{attribute 'linkalways'} 
{attribute 'no_explicit_call' := 'This FB is a CLASS and must be accessed using methods or properties'}
{attribute 'enable_dynamic_creation'}
FUNCTION_BLOCK DefaultHomingBuilder IMPLEMENTS I_HomingBuilder, I_PositioningHomingBuilder, I_DefaultHomingBuilder
VAR
	_axis : I_Axis;
	_position : LREAL;
	_options : ST_HomingOptions;
	_cam : REFERENCE TO BOOL;
END_VAR

METHOD BuildDefaultHomingCommand : I_HomingCommand
VAR
	pCmd : POINTER TO HomingCommand;
	cmd : I_HomingCommand;
END_VAR
pCmd := __NEW(HomingCommand(
	axis := _axis,
	position := _position,
	mode := HomingMode.Default,
	options := _options,
	cam := _cam
));
BuildDefaultHomingCommand := pCmd^;
END_METHOD

METHOD BuildDirectHomingCommand : I_HomingCommand
VAR
	pCmd : POINTER TO HomingCommand;
	cmd : I_HomingCommand;
	null : BOOL;
END_VAR
pCmd := __NEW(HomingCommand(
	axis := _axis,
	position := _position,
	mode := HomingMode.Direct,
	options := _options,
	cam := null
));
BuildDirectHomingCommand := pCmd^;
END_METHOD

METHOD BuildForceCalibrationCommand : I_HomingCommand
VAR
	pCmd : POINTER TO HomingCommand;
	cmd : I_HomingCommand;
	null : BOOL;
END_VAR
pCmd := __NEW(HomingCommand(
	axis := _axis,
	position := _position,
	mode := HomingMode.ForceCalibration,
	options := _options,
	cam := null
));
BuildForceCalibrationCommand := pCmd^;
END_METHOD

METHOD BuildResetCalibrationCommand : I_HomingCommand
VAR
	pCmd : POINTER TO HomingCommand;
	cmd : I_HomingCommand;
	null : BOOL;
END_VAR
pCmd := __NEW(HomingCommand(
	axis := _axis,
	position := _position,
	mode := HomingMode.ResetCalibration,
	options := _options,
	cam := null
));
BuildResetCalibrationCommand := pCmd^;
END_METHOD

METHOD Cam : I_DefaultHomingBuilder
VAR_INPUT
	value : REFERENCE TO BOOL;
END_VAR
_cam REF= value;
Cam := THIS^;
END_METHOD

METHOD ClearLag : I_PositioningHomingBuilder
_options.ClearPositionLag := TRUE;
ClearLag := THIS^;
END_METHOD

METHOD FB_init : BOOL
VAR_INPUT
	bInitRetains : BOOL; // if TRUE, the retain variables are initialized (warm start / cold start)
	bInCopyCode : BOOL;  // if TRUE, the instance afterwards gets moved into the copy code (online change)
	axis : I_Axis;
END_VAR
_axis := axis;
END_METHOD

METHOD KeepLag : I_PositioningHomingBuilder
_options.ClearPositionLag := FALSE;
KeepLag := THIS^;
END_METHOD

METHOD Position : I_PositioningHomingBuilder
VAR_INPUT
	value : LREAL;
END_VAR
_position := value;
Position := THIS^;
END_METHOD

METHOD ReferenceMode : I_DefaultHomingBuilder
VAR_INPUT
	value : EncoderReferenceMode;
END_VAR
_options.ReferenceMode := value;
ReferenceMode := THIS^;
END_METHOD

METHOD SearchDirection : I_DefaultHomingBuilder
VAR_INPUT
	value : Direction;
END_VAR
_options.SearchDirection := value;
SearchDirection := THIS^;
END_METHOD

METHOD SearchVelocity : I_DefaultHomingBuilder
VAR_INPUT
	value	: LREAL;
END_VAR
_options.SearchVelocity := value;
SearchVelocity := THIS^;
END_METHOD

METHOD SyncDirection : I_DefaultHomingBuilder
VAR_INPUT
	value : Direction;
END_VAR
_options.SyncDirection := value;
SyncDirection := THIS^;
END_METHOD

METHOD SyncVelocity : I_DefaultHomingBuilder
VAR_INPUT
	value : LREAL;
END_VAR
_options.SyncVelocity := value;
SyncVelocity := THIS^;
END_METHOD

END_FUNCTION_BLOCK

(* stored: Version 1.1.0.1, ProductVersion 3.1.4024.12
   POU DefaultHomingBuilder: Id {f8c09a37-3872-4c76-9ad7-78df88afe57e}, SpecialFunc None
   Folder Builders: Id {acb2335d-7e37-4096-bebb-815ba4dfd342}
   Folder Property Setters: Id {4a604d78-4592-4df9-b8bc-f4f35e4ceb1e}
   Method BuildDefaultHomingCommand: Id {60cdb31b-248f-4a5e-a6c7-53ec1d7013c8}
   Method BuildDirectHomingCommand: Id {dd77a1a7-1a20-4bf4-a585-a10b4cce35ce}
   Method BuildForceCalibrationCommand: Id {1fed35d2-767b-4b68-ba0c-a819755b2e4c}
   Method BuildResetCalibrationCommand: Id {7a12bfc3-4c4b-44ca-99fa-53cd3375db3e}
   Method Cam: Id {b59a248a-e19b-478f-a37b-a81f0685cd4d}
   Method ClearLag: Id {fc0cb63b-b614-4397-a1e5-160469549e44}
   Method FB_init: Id {f0140b19-f229-4aba-97db-41810c48608c}
   Method KeepLag: Id {61d79078-56a0-4b74-a1b7-95dea3c1eab5}
   Method Position: Id {2a021c4c-3804-43d5-9d7b-1d9e6d7a80a4}
   Method ReferenceMode: Id {04a1bc16-ae5b-4c82-8fbd-81d5e8756c2f}
   Method SearchDirection: Id {52af2548-e1fc-4cc4-814c-5c68f8ecbf54}
   Method SearchVelocity: Id {72bab1cd-20d2-4cac-a28e-2b0ac440d737}
   Method SyncDirection: Id {5172015f-cffd-48df-ba6e-c06d8d8cd959}
   Method SyncVelocity: Id {8403b227-9b1f-492f-bacd-40076f055bf2} *)
